// TIA Portal V16 export
// export: Created 2024-09-05T17:39:14.6686231Z, ExportSetting WithDefaults, DisplayName Totally Integrated Automation Portal, DisplayVersion V16 Update 6, DisplayName TIA Portal Version Control Interface, DisplayVersion V16 Update 2, DisplayName TIA Portal Openness, DisplayVersion V16 Update 6, DisplayName STEP 7 Professional, DisplayVersion V16 Update 6, DisplayName STEP 7 Safety, DisplayVersion V16, DisplayName WinCC Advanced, DisplayVersion V16 Update 6
FUNCTION "FC_ShiftIntervalCompare" : Void   // FC5010, LAD
{ S7_Optimized_Access := 'TRUE' }
VERSION : 0.1
// stored: AutoNumber false, IsIECCheckEnabled false, SetENOAutomatically false, UDAEnableTagReadback false
   VAR_INPUT
      iRequiredShiftNumber : UInt;
      iShiftStartTime : Time_Of_Day;
      iShiftEndTime : Time_Of_Day;
      iActualTime : Time_Of_Day;
   END_VAR
   VAR_IN_OUT
      iqShiftNumber : UInt;
   END_VAR
   VAR_TEMP
      midnight_time : Time_Of_Day;
      morning_time : Time_Of_Day;
      interval_in_two_days : Bool;
   END_VAR
BEGIN

REGION Network 1: Shift interval compare
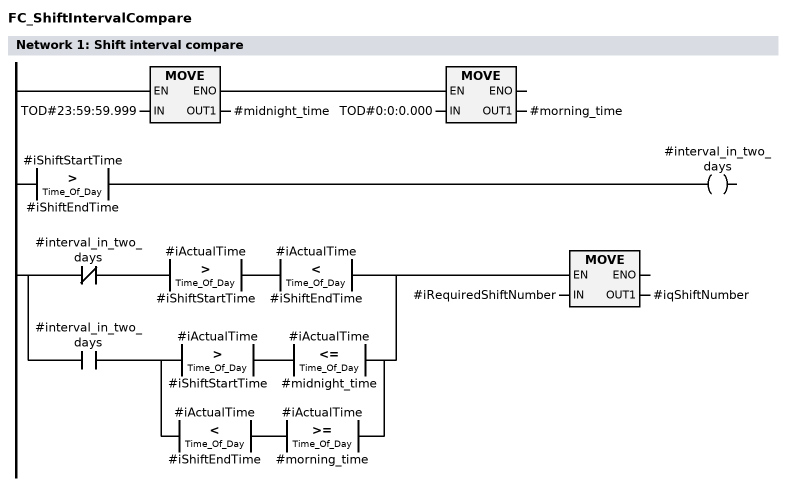
   RUNG wire#powerrail
      Move(in := TOD#23:59:59.999, out1 => #midnight_time)
      Move(in := TOD#0:0:0.000, out1 => #morning_time)
   END_RUNG
   RUNG wire#powerrail
      { S7_Templates := "SrcType := Time_Of_Day" } GT_Contact(in1 := #iShiftStartTime, in2 := #iShiftEndTime)
      Coil( #interval_in_two_days )
   END_RUNG
   RUNG wire#powerrail
      I_Contact( #interval_in_two_days )
      { S7_Templates := "SrcType := Time_Of_Day" } GT_Contact(in1 := #iActualTime, in2 := #iShiftStartTime)
      { S7_Templates := "SrcType := Time_Of_Day" } LT_Contact(in1 := #iActualTime, in2 := #iShiftEndTime)
      wire#w1
      Move(in := #iRequiredShiftNumber, out1 => #iqShiftNumber)
   END_RUNG
   RUNG wire#powerrail
      Contact( #interval_in_two_days )
      wire#w2
      { S7_Templates := "SrcType := Time_Of_Day" } GT_Contact(in1 := #iActualTime, in2 := #iShiftStartTime)
      { S7_Templates := "SrcType := Time_Of_Day" } LE_Contact(in1 := #iActualTime, in2 := #midnight_time)
   END_RUNG wire#w1
   RUNG wire#w2
      { S7_Templates := "SrcType := Time_Of_Day" } LT_Contact(in1 := #iActualTime, in2 := #iShiftEndTime)
      { S7_Templates := "SrcType := Time_Of_Day" } GE_Contact(in1 := #iActualTime, in2 := #morning_time)
   END_RUNG wire#w1
   // the same network as SCL:
   #midnight_time := TOD#23:59:59.999;
   #morning_time := TOD#0:0:0.000;
   #interval_in_two_days := #iShiftStartTime > #iShiftEndTime;
   IF (NOT #interval_in_two_days AND (#iActualTime > #iShiftStartTime) AND (#iActualTime < #iShiftEndTime)) OR (#interval_in_two_days AND (((#iActualTime > #iShiftStartTime) AND (#iActualTime <= #midnight_time)) OR ((#iActualTime < #iShiftEndTime) AND (#iActualTime >= #morning_time)))) THEN
       #iqShiftNumber := #iRequiredShiftNumber;
   END_IF;
END_REGION
END_FUNCTION
